# EPICS substitutions: epicsApp/K18MonitorApp/Db/GL840_RC.substitutions
# GL840_AFT substitutions file
# ch   :  form 1 to 7

file "db/GL840_RC.template" {
   { name=RC:X+:TEMP,  ch=1,  ASLO=1, ESLO=0.005, EOFF=0 }
   { name=RC:X-:TEMP,  ch=2,  ASLO=1, ESLO=0.005, EOFF=0 }
}
